FUNCTION_BLOCK TcA2B2Kitten
VAR_INPUT
END_VAR
VAR_OUTPUT
END_VAR
VAR
	_ConnectCommand: 		PLCopenCommand;
	_httpClient:			FB_IotHttpClient;
	_httpRequest:			FB_IotHttpRequest;
	_httpRequestHeader:		FB_IotHttpHeaderFieldMap;
	bSendGet:				BOOL;
	connectNow: 			BOOL;
	requestNow: 			BOOL;
	sContent				: STRING(511);
END_VAR



_httpClient.sHostName := '192.168.56.1';
_httpClient.nHostPort := 80;
_httpClient.bKeepAlive := TRUE;
_httpClient.stTLS.bNoServerCertCheck:=TRUE;
_httpClient.tConnectionTimeout := T#10S;

IF connectNow THEN
	_httpClient.Execute();
END_IF



IF _httpClient.bConnected AND requestNow THEN
	//_httpRequest.eCompressionMode := ;
	//_httpRequest.sContentType := ;
	
	_httpRequestHeader.AddField('accept', 'application/hal+json;v=2.0', FALSE);
	_httpRequestHeader.AddField('authorization', 'Basic RGVmYXVsdCBVc2VyOnJvYm90aWNz', TRUE);
	
	_httpRequest.SendRequest(sUri:='/rw/rapid/execution', fbClient:=_httpClient, eRequestType:=ETcIotHttpRequestType.HTTP_Get, pContent:=ADR(sContent), nContentSize:=SIZEOF(sContent), fbHeader:=_httpRequestHeader);

	requestNow := FALSE;
END_IF

METHOD Connect : BOOL
VAR_INPUT
	ip:	DINT;
	status: IPLCopenCall;
END_VAR









IF status = 0 THEN
	_ConnectCommand.Execute := 1;
ELSE
	status.Start(_ConnectCommand);
END_IF
END_METHOD

METHOD Connect_Impl : BOOL
VAR_INPUT
END_VAR
END_METHOD

METHOD Cyclic : BOOL
VAR_INPUT
END_VAR

(*
IF _ConnectCommand.Consume THEN
	;//TempSetPoint := 350; //set the oven temp set point
	
END_IF

Connect_Impl();

IF connected THEN 
	_ConnectCommand.Finished();
END_IF

_ConnectCommand.Execute := 0;
*)
END_METHOD

METHOD GetRobotState : BOOL
VAR_INPUT
	call: PLCopenCall;
END_VAR
END_METHOD

END_FUNCTION_BLOCK

(* stored: Version 1.1.0.1, ProductVersion 3.1.4024.12
   POU TcA2B2Kitten: Id {ea1fde4a-6390-43d8-ae6c-e82c42f674c2}, SpecialFunc None
   Method Connect: Id {e7faa834-d121-4df0-9a35-0dedcf979687}
   Method Connect_Impl: Id {d93b10d7-23fa-4f77-88b2-ba9c5838001e}
   Method Cyclic: Id {e891cab9-f69d-4866-ae67-7ef69a98b4aa}
   Method GetRobotState: Id {6fdc1b90-83fc-42a7-8e4c-63e16e67acec} *)
